FUNCTION_BLOCK ButtonNO IMPLEMENTS I_Button
VAR
	bInput	AT%I*	: BOOL;
	rtInput			: R_TRIG;
END_VAR

PROPERTY IsPressed : BOOL
GET
IsPressed := bInput;
END_GET
END_PROPERTY

PROPERTY IsReleased : BOOL
GET
IsReleased := NOT IsPressed;
END_GET
END_PROPERTY

PROPERTY RisingTrigger : BOOL
GET
rtInput(CLK := IsPressed);

RisingTrigger := rtInput.Q;
END_GET
END_PROPERTY

END_FUNCTION_BLOCK

(* stored: Version 1.1.0.1
   POU ButtonNO: Id {9648fb86-2586-4f86-af45-2503960afbd3}, SpecialFunc None
   Property IsPressed: Id {399b64f0-f69f-44c3-93ed-d0388813c38c}
   Get Get: Id {d52789a7-20c7-4c29-a7bf-18c548688d6a}
   Property IsReleased: Id {9c52060c-62d5-4c3b-bcb0-25b425f1e19d}
   Get Get: Id {a4853a07-d314-41a5-a91f-7e59d26a4507}
   Property RisingTrigger: Id {fee4ae38-22e9-4ec8-a98c-8370d3268195}
   Get Get: Id {d844dd31-6472-4536-898c-c8c68b35ff16} *)
